FUNCTION_BLOCK FB_Base EXTENDS FB_BasePart IMPLEMENTS I_Elementinformation, I_TestInterface
(*
 @details
 The FB_Base is the base function block of the.
 @usage
 The function block works like this or like that.
 also there are multiline stuff possible
*)
VAR
	//Elementinformation
  _bCodeActive 						: BOOL; // this does that or those
	_bEnableCode              			: BOOL;  (* other possible comment *)          

	{attribute 'hide'}                							
	_bUseParentEnableCode				: BOOL; (*** other possible comment *)
	
    _bEnableAlarm         				: BOOL := TRUE;
    {attribute 'hide'}
	_bUseParentEnableAlarm				: BOOL;   
		
    _eSimulation      					: E_SimulationMode := E_SimulationMode.simOff;
    {attribute 'hide'}
	_bUseParentSimulation				: BOOL;
	
	_bReset								: BOOL;
    {attribute 'hide'}
	_bUseParentReset					: BOOL;
	
	_nParentNumber						: INT;
    {attribute 'hide'}
	_bUseParentNumber					: BOOL;
	
	_sParentName						: STRING(Par_Core.C_nLengthOfParentName);
    {attribute 'hide'}
	_bUseParentName						: BOOL;	
	
    _sDesignationName     				: STRING(Par_Core.C_nLengthOfDesignationName);      
	
	_bError								: BOOL;
	
    {attribute 'hide'}
    _iParentInformation 				: I_ElementInformation;												
    {attribute 'hide'}
    _eCodeExecution 					: E_CodeExecutionMode; 										
	
	// Logging
	{attribute 'hide'}
	_LogCollector						: FB_LogCollector;
    {attribute 'hide'}	        		
	_BaseLogger							: FB_Log := (logCollector := _LogCollector);
END_VAR

VAR_STAT
	{attribute 'hide'}
	_bLicenseOk 							: BOOL := TRUE; // static class variable, access to all fb
END_VAR

METHOD PROTECTED _ConfigureAlarm : BOOL;
(***********************************************************************************
* @brief Description : Gets called in enabling
* @return None
************************************************************************************)
// Call update once to enable/disableAlarms
_UpdateAlarm();
_BaseLogger.Info(sMsg := 'Alarms configured').Send();
_ConfigureAlarm := TRUE;
END_METHOD

METHOD PROTECTED _ConfigureHmi : BOOL;
// gets called in enabling
// do some elementmgr magic
_BaseLogger.Debug(sMsg := 'HMI configured').Send();
_ConfigureHmi := TRUE;
END_METHOD

METHOD PROTECTED _Disabling : BOOL;
(***********************************************************************************
* @brief Description : Logic which disables the function block
* @return BOOL 1 = Disabling completed
************************************************************************************)
_ResetError(); // call reset method
_Disabling := _ConfigureAlarm() AND _ConfigureHmi();
END_METHOD

METHOD PROTECTED _Enabling : BOOL
_ResetError(); // call reset method
_Enabling := _ConfigureAlarm() AND _ConfigureHmi();
END_METHOD

METHOD PRIVATE _GetParentInformation
IF _iParentInformation <> 0 THEN
	IF _bUseParentEnableAlarm 	THEN _bEnableAlarm 		:= _iParentInformation.EnableAlarm; 	END_IF
	IF _bUseParentEnableCode 	THEN _bEnableCode 		:= _iParentInformation.EnableCode; 		END_IF
	IF _bUseParentReset 		THEN _bReset 			:= _iParentInformation.Reset; 			END_IF
	IF _bUseParentSimulation 	THEN _eSimulation 		:= _iParentInformation.Simulation; 		END_IF
	IF _bUseParentName 	THEN _sParentName 		:= _iParentInformation.ParentName; 		END_IF
	IF _bUseParentNumber 	THEN _nParentNumber 	:= _iParentInformation.ParentNumber; 	END_IF
END_IF
END_METHOD

METHOD PROTECTED _MainGeneral






_UpdateAlarm();
_UpdateHmi();
IF _bReset THEN
	_ResetError();
END_IF
END_METHOD

METHOD PROTECTED _ResetError
(***********************************************************************************
* @brief Description : Gets called if bReset is true, in enabling,disabling and maingeneral
* @return None
************************************************************************************)
// do some things








_UpdateAlarm();
_BaseLogger.Debug(sMsg := 'Reset triggered').Send();
END_METHOD

METHOD PROTECTED _SetError
(***********************************************************************************
* @brief Description : gets called by update Alarm, used to set the error bit
* @return None
************************************************************************************)
// set the function block error bit
_bError := FALSE;
END_METHOD

METHOD PROTECTED _UpdateAlarm
(***********************************************************************************
* @brief Description : Call of all alarm function blocks
* @return None
************************************************************************************)
//// Example







// Call error collection method
_SetError();
END_METHOD

METHOD PROTECTED _UpdateHmi
(***********************************************************************************
* @brief Description : Method to update the HMI interface
* @return None
************************************************************************************)
// copy all internal parameters to the HMI interface
END_METHOD

METHOD PUBLIC CyclicGeneral

VAR_INST
	{attribute 'hide'}
	_EnableCodeLogger 		: FB_LogVar := (LogCollector := LogCollector);
	{attribute 'hide'}
	_EnableAlarmLogger 		: FB_LogVar := (LogCollector := LogCollector);
	{attribute 'hide'}
	_CodeActiveLogger 		: FB_LogVar := (LogCollector := LogCollector);
	{attribute 'hide'}
	_DesignationNameLogger 	: FB_LogVar := (LogCollector := LogCollector);
	{attribute 'hide'}
	_SimulationLogger 		: FB_LogVar := (LogCollector := LogCollector);
	{attribute 'hide'}
	_ParentNameLogger 		: FB_LogVar := (LogCollector := LogCollector);
	{attribute 'hide'}
	_ParentNumberLogger 	: FB_LogVar := (LogCollector := LogCollector);
END_VAR
_GetParentInformation();
_EnableCodeLogger.OnChange(_bEnableCode);

CASE _eCodeExecution OF
    E_CodeExecutionMode.enable:
        IF _Enabling() THEN
            _eCodeExecution := E_CodeExecutionMode.cyclic;
        END_IF

    E_CodeExecutionMode.cyclic:
        IF NOT _bEnableCode OR NOT _bLicenseOk THEN
            _eCodeExecution := E_CodeExecutionMode.disable;
        END_IF

    E_CodeExecutionMode.disable:
        IF _Disabling() THEN
            _eCodeExecution := E_CodeExecutionMode.undefined;
        END_IF

    E_CodeExecutionMode.undefined:
        IF _bEnableCode AND _bLicenseOk THEN		
            _eCodeExecution := E_CodeExecutionMode.enable;
        END_IF
END_CASE

_bCodeActive := _eCodeExecution = E_CodeExecutionMode.cyclic;
_CodeActiveLogger.OnChange(_bCodeActive);

IF _bCodeActive THEN
	_DesignationNameLogger.OnChange(_sDesignationName);
	_ParentNameLogger.OnChange(_sParentName);
	_ParentNumberLogger.OnChange(_nParentNumber);
	_EnableAlarmLogger.OnChange(_bEnableCode);
	_SimulationLogger.OnChange(_eSimulation);
    _MainGeneral();
END_IF
END_METHOD

PROPERTY DesignationName : String(Par_Core.C_nLengthOfDesignationName)
GET
DesignationName := THIS^._sDesignationName;
END_GET
SET
THIS^._sDesignationName := DesignationName;
END_SET
END_PROPERTY

PROPERTY EnableAlarm : BOOL
GET
EnableAlarm := THIS^._bEnableAlarm;
END_GET
SET
_bUseParentEnableAlarm := FALSE;
THIS^._bEnableAlarm := EnableAlarm;
END_SET
END_PROPERTY

PROPERTY EnableCode : Bool
GET
EnableCode := THIS^._bCodeActive;
END_GET
SET
_bUseParentEnableCode := FALSE;
THIS^._bEnableCode := EnableCode;
END_SET
END_PROPERTY

PROPERTY Error : BOOL
GET
Error := THIS^._bError;
END_GET
END_PROPERTY

PROPERTY LogCollector : REFERENCE TO FB_LogCollector
GET
LogCollector REF= _LogCollector;
END_GET
END_PROPERTY

PROPERTY Parent : I_ElementInformation
SET
_iParentInformation 			:= Parent;
// Reset all information selectors
_bUseParentReset 			:= TRUE;
_bUseParentEnableCode 		:= TRUE;
_bUseParentEnableAlarm 		:= TRUE;
_bUseParentSimulation 		:= TRUE;
_bUseParentNumber		:= TRUE;
_bUseParentName		:= True;
END_SET
END_PROPERTY

PROPERTY ParentName : STRING(Par_Core.C_nLengthOfParentName)
GET
ParentName := THIS^._sParentName;
END_GET
SET
_bUseParentName := FALSE;
THIS^._sParentName := ParentName;
END_SET
END_PROPERTY

PROPERTY ParentNumber : INT
GET
ParentNumber := THIS^._nParentNumber;
END_GET
SET
_bUseParentNumber := FALSE;
THIS^._nParentNumber := ParentNumber;
END_SET
END_PROPERTY

PROPERTY Reset : BOOL
GET
Reset := THIS^._bReset;
END_GET
SET
_bUseParentReset := FALSE;
THIS^._bReset := Reset;
END_SET
END_PROPERTY

PROPERTY Simulation : E_SimulationMode
GET
Simulation := THIS^._eSimulation;
END_GET
SET
_bUseParentSimulation := FALSE;
THIS^._eSimulation := Simulation;
END_SET
END_PROPERTY

END_FUNCTION_BLOCK

(* stored: Version 1.1.0.1, ProductVersion 3.1.4024.12
   POU FB_Base: Id {ae258f57-8349-41d4-9dcd-5e11bbba79e4}, SpecialFunc None
   Folder External: Id {644b7fe0-1b81-4012-ae47-0a9d6a4ddaf0}
   Folder Cyclic: Id {66851ef5-4a16-4212-bc1e-020ddbb0600e}
   Folder ElementInformation: Id {299da64f-9e3e-4f49-a9ed-4e21ddaacf78}
   Folder Internal: Id {0dfa9513-08d8-4087-9bfa-06d9c0f2a5de}
   Folder Alarm: Id {72c74cb0-177c-4495-9f02-b2386fee407f}
   Folder Error: Id {e2fe0268-cb79-417f-9c08-d6d2f4b840f0}
   Folder Hmi: Id {a04651d6-80a6-4d9e-a265-747bcd93077b}
   Folder Logging: Id {292e455d-6e5a-4ade-9ed2-b549b8e0f798}
   Method _ConfigureAlarm: Id {45a3ec5b-7241-4a4c-967e-684dee223ad7}
   Method _ConfigureHmi: Id {bee58f22-9a7a-438a-9923-d7cc2a50e47d}
   Method _Disabling: Id {ca184a1d-ad07-49e1-8807-681f6213d1e5}
   Method _Enabling: Id {1941c1a7-98e5-42d3-b1ff-31a93388b95a}
   Method _GetParentInformation: Id {7e22c7e0-5e4f-4d4a-9c50-0abb2847914b}
   Method _MainGeneral: Id {203b172e-859f-4316-af01-0872fbbb1c80}
   Method _ResetError: Id {90906135-6609-43a9-b296-a6983ebe86e2}
   Method _SetError: Id {90272852-62aa-4bdd-b315-5ac2ae233479}
   Method _UpdateAlarm: Id {ed6b3f20-7366-4f42-ac50-4b23411a20cd}
   Method _UpdateHmi: Id {9503ce37-dc79-4f37-aacc-ed2eafc83780}
   Method CyclicGeneral: Id {3c5c321f-6670-46a8-bbc3-149ff338d692}
   Property DesignationName: Id {2b07be22-2703-43af-8b6b-38139b620086}
   Get Get: Id {52ec2361-f01a-4ef6-80d0-fbb75289521f}
   Set Set: Id {d77c8f5d-0989-406f-aad7-00725eae2b55}
   Property EnableAlarm: Id {83a03a7a-d617-45a2-867b-dbfbeb2771b0}
   Get Get: Id {194df314-021a-4578-963f-c5c1ecb85b34}
   Set Set: Id {7f1792ff-97a7-4839-a232-3000f19224b4}
   Property EnableCode: Id {15f2624c-0669-4454-8048-44a82b4da53a}
   Get Get: Id {c1e9d95f-75d8-416d-88ab-db03cc0a14cb}
   Set Set: Id {46202e93-ab20-459e-8ad6-3cf87a7696fa}
   Property Error: Id {70f833c0-c50e-441d-aa7c-9df706ffab5b}
   Get Get: Id {8f2619b3-5004-4d16-99bb-0e18731ea4c9}
   Property LogCollector: Id {adfe944a-f435-407a-8921-dc4caeb31b01}
   Get Get: Id {c65275c8-c826-40ef-a5d0-9540de438477}
   Property Parent: Id {2d0fedf9-593e-4499-968d-e6045e383501}
   Set Set: Id {29ecbc33-84a1-4663-b64e-08a3d1480ed3}
   Property ParentName: Id {56e98454-019c-4dc6-8bdf-2203b95184c7}
   Get Get: Id {2cf50430-f590-47bd-960d-daabac11a2c5}
   Set Set: Id {c815d856-2159-4a4b-9e86-da0d8ba172f7}
   Property ParentNumber: Id {99503c9f-d3be-48e6-bcc4-464a22849af2}
   Get Get: Id {77ae15b3-abb9-40a4-8fd8-045a7795910b}
   Set Set: Id {c16baaac-626a-4708-9ab9-f32cc02c3217}
   Property Reset: Id {18e3ae02-8020-43c1-8ac3-b42813f58858}
   Get Get: Id {650b18b0-3694-4de3-9ff2-daf2f64740cd}
   Set Set: Id {76ed96c1-77e6-4944-a950-8f352bcb0fe3}
   Property Simulation: Id {6a62df8c-b165-4c7f-9010-807c3f15f925}
   Get Get: Id {52e0e525-56e4-44b6-a857-e6145ff02d01}
   Set Set: Id {a0098d24-7d7e-4fec-8f41-404a01da5430} *)
